(* IEC 61131-3 sources: AXOpen/src/components.pneumatics/app/src/Documentation/IO, 6 files *)

(* ---- HwInputs.st ---- *)
TYPE
	{S7.extern=ReadWrite}
	HwInputs : STRUCT
		ET200SP_DI_8x24VDC_ST_V1_1_1 AT %B0 : BYTE;
	END_STRUCT;
END_TYPE

(* ---- HwOutputs.st ---- *)
TYPE
	HwOutputs : STRUCT
		ET200SP_DQ_8x24VDC_0_5A_ST_V1_1_1 AT %B0 : BYTE;
	END_STRUCT;
END_TYPE

(* ---- PlcInputs.st ---- *)
TYPE
	PlcInputs : STRUCT
		ET200SP_DI_8x24VDC_ST_V1_1_1 : BYTE;
	END_STRUCT;
END_TYPE

(* ---- PlcOutputs.st ---- *)
TYPE
	PlcOutputs : STRUCT
		ET200SP_DQ_8x24VDC_0_5A_ST_V1_1_1 : BYTE;
	END_STRUCT;
END_TYPE

(* ---- CopyInputs.st ---- *)
FUNCTION CopyInputs
	VAR_EXTERNAL
		HwInputs : HwInputs;
		PlcInputs : PlcInputs;
	END_VAR
	PlcInputs.ET200SP_DI_8x24VDC_ST_V1_1_1 := HwInputs.ET200SP_DI_8x24VDC_ST_V1_1_1;
END_FUNCTION

(* ---- CopyOutputs.st ---- *)
FUNCTION CopyOutputs
	VAR_EXTERNAL
		HwOutputs : HwOutputs;
		PlcOutputs : PlcOutputs;
	END_VAR
	HwOutputs.ET200SP_DQ_8x24VDC_0_5A_ST_V1_1_1 := PlcOutputs.ET200SP_DQ_8x24VDC_0_5A_ST_V1_1_1;
END_FUNCTION
